FUNCTION F_ComputeSInt32Size : UDINT
VAR_INPUT
    anyDint : ANY;
END_VAR
VAR
    nValue  : DINT;
END_VAR

memcpy(destAddr:= ADR(nValue), srcAddr:= anyDint.pValue, n:= MIN(TO_UDINT(anyDint.diSize), SIZEOF(nValue)));
F_ComputeSInt32Size := F_ComputeRawVarint32Size(F_EncodeZigZag32(nValue));

END_FUNCTION

(* stored: Version 1.1.0.1
   POU F_ComputeSInt32Size: Id {d2cfb765-286e-450e-89e8-1f039ec738be}, SpecialFunc None *)
